// TIA Portal V19 export
VAR_GLOBAL   // PLC tag table "D15"
   D15_Lp_EntryReq_LB222 AT %Q109.5 : Bool;   // 241SH1
   D15_Lp_SafetyReset_LB222 AT %Q109.6 : Bool;   // 241SH2
   D15_Pb_EntryReq_LB222 AT %I108.4 : Bool;   // 241SH1
   D15_Pb_SafetyReset_LB222 AT %I108.5 : Bool;   // 241SH2
   D15_Comando_Elettroserratura AT %Q109.4 : Bool;   // 24102
   D15_Cancello_Chiuso AT %I108.2 : Bool;   // 24101
   D15_Cancello_Bloccato AT %I108.3 : Bool;   // 24103
   D15_Ls_Os1 AT %I1079.2 : Bool;   // 106DI2 - 241A1
   D15_Ls_Os2 AT %I1079.6 : Bool;   // 106DI6 - 241A1
END_VAR
